KUKA KRL data list: coin2.dat

&ACCESS RVP
&REL 9
&PARAM DISKPATH = KRC:\R1\3dTisk
&PARAM TEMPLATE = C:\KRC\Roboter\Template\ExpertVorgabe
&PARAM EDITMASK = *
DEFDAT  coin2
;FOLD EXTERNAL DECLARATIONS;%{PE}%MKUKATPBASIS,%CEXT,%VCOMMON,%P
;FOLD BASISTECH EXT;%{PE}%MKUKATPBASIS,%CEXT,%VEXT,%P
EXT  BAS (BAS_COMMAND  :IN,REAL  :IN )
DECL INT SUCCESS
;ENDFOLD (BASISTECH EXT)
;FOLD USER EXT;%{E}%MKUKATPUSER,%CEXT,%VEXT,%P
;Make your modifications here

;ENDFOLD (USER EXT)
;ENDFOLD (EXTERNAL DECLARATIONS)
DECL BASIS_SUGG_T LAST_BASIS={POINT1[] "P2                      ",POINT2[] "P2                      ",CP_PARAMS[] "CPDAT2                  ",PTP_PARAMS[] "PDAT0                   ",CONT[] "                        ",CP_VEL[] "0.5                     ",PTP_VEL[] "100                     ",SPL_NAME[] "S0                      "}
DECL E6POS XP1={X 358.691589,Y 200.225403,Z -0.0274270307,A 0.0223432798,B -0.00957637932,C -0.0179978702,S 6,T 27,E1 0.0,E2 0.0,E3 0.0,E4 0.0,E5 0.0,E6 0.0}
DECL FDAT FP1={TOOL_NO 8,BASE_NO 8,IPO_FRAME #BASE,POINT2[] " ",TQ_STATE FALSE}
DECL LDAT LCPDAT1={VEL 2.0,ACC 100.0,APO_DIST 100.0,APO_FAC 50.0,AXIS_VEL 100.0,AXIS_ACC 100.0,ORI_TYP #VAR,CIRC_TYP #BASE,JERK_FAC 50.0,GEAR_JERK 50.0,EXAX_IGN 0}
DECL LDAT LCPDAT2={VEL 2.0,ACC 100.0,APO_DIST 100.0,APO_FAC 50.0,AXIS_VEL 100.0,AXIS_ACC 100.0,ORI_TYP #VAR,CIRC_TYP #BASE,JERK_FAC 50.0,GEAR_JERK 50.0,EXAX_IGN 0}
DECL E6POS XP2={X 358.691589,Y 200.225403,Z -0.0274270307,A 0.0223432798,B -0.00957637932,C -0.0179978702,S 6,T 27,E1 0.0,E2 0.0,E3 0.0,E4 0.0,E5 0.0,E6 0.0}
DECL FDAT FP2={TOOL_NO 8,BASE_NO 8,IPO_FRAME #BASE,POINT2[] " ",TQ_STATE FALSE}
ENDDAT
